INTERFACE I_NAME

PROPERTY Name : STRING
GET
END_GET
SET
END_SET
END_PROPERTY

METHOD NUM : INT
VAR_INPUT
END_VAR
END_METHOD

END_INTERFACE

(* stored: Version 1.1.0.1, ProductVersion 3.1.4024.3
   Itf I_NAME: Id {1577b5ca-943e-47e7-be8c-425ad164604b}
   Property Name: Id {3b820094-dc39-4468-b76c-cdf826009ebd}
   Get Get: Id {709566d5-1830-4eba-a17f-583e4484bf19}
   Set Set: Id {05e10362-1841-4475-9b45-9e616eb79680}
   Method NUM: Id {3707bedd-a78d-4f50-a9b3-d91374717364} *)
